{attribute 'qualified_only'}
{attribute 'strict'}
TYPE Command :
(
	Stop 		:= 0,
	Abort 		:= 1,
	Executing 	:= 2,
	Hold 		:= 3,
	Reset 		:= 4
);
END_TYPE

(* stored: Version 1.1.0.1, ProductVersion 3.1.4024.6
   DUT Command: Id {c1f1d2c9-8926-4429-8b54-eb7c4f63f81a} *)
